{attribute 'qualified_only'}
{attribute 'strict'}
{attribute 'to_string'}
TYPE EStrategyStates :
(
	none := 0,
	ready := 1,
	running := 2,
	halting := 3,
	halted := 4,
	done := 5
) USINT;
END_TYPE

(* stored: Version 1.1.0.1
   DUT EStrategyStates: Id {0fed0be0-7395-419a-9b57-41fdfb27e845} *)
